# EPICS substitutions: lensApp/Db/fixedlimit.substitutions
file fixedlimit.tpl-db
{
    {
        LOCATION   = $(LOCATION)
        LIMIT      = $(LIMIT)
        LOW_LIMIT  = $(LOW_LIMIT)
        HIGH_LIMIT = $(HIGH_LIMIT)
    }
}
file limit.tpl-db
{
    {
        LOCATION = $(LOCATION)
        LIMIT    = $(LIMIT)
    }
}
